// TIA Portal V15.1 export
// export: Created 2024-05-17T05:38:35.0496997Z, ExportSetting WithDefaults, DisplayName Totally Integrated Automation Portal, DisplayVersion V15.1 Update 5, DisplayName TIA Portal Openness, DisplayVersion V15.1 Update 5, DisplayName SINAMICS Startdrive Advanced, DisplayVersion V15.1, DisplayName G130, G150, S120, S150, SINAMICS MV, S210, DisplayVersion V15.1, DisplayName G110M, G120, G120C, G120D, G120P, DisplayVersion V15.1, DisplayName STEP 7 Professional, DisplayVersion V15.1 Update 5, DisplayName STEP 7 Safety, DisplayVersion V15.1, DisplayName WinCC Professional, DisplayVersion V15.1 Update 5, DisplayName SIMATIC Visualization Architect, DisplayVersion V15.1
FUNCTION_BLOCK "LProcPid"   // FB1713, FBD
TITLE = LProcPid
{ S7_Optimized_Access := 'FALSE' }
AUTHOR : VCC
FAMILY : ProcEq
NAME : Pid
VERSION : 0.1
// ================================================================================
// The Process Value is controlled by the Pid controller.
// ================================================================================
// stored: AutoNumber false, IsIECCheckEnabled false, SetENOAutomatically False, UDAEnableTagReadback false
   VAR_INPUT
      I_CYCLE { ExternalAccessible := 'False'; ExternalVisible := 'False'; ExternalWritable := 'False'} : Time;   // Sample time
      H_TI : Time;   // Pid Reset time
      H_TD : Time;   // Pid Derivative time
      I_Manual_Value { ExternalAccessible := 'False'; ExternalVisible := 'False'; ExternalWritable := 'False'} : Real;   // Pid Setpoint Manual
      I_SP_Auto : Real;   // Pid Setpoint for controller
      I_PV_PID : Real;   // Pid Process value
      H_GAIN : Real;   // Pid Proportional Gain
      H_DEADB_W : Real;   // Pid Deadband width
      H_LMN_HLM : Real := 100.0;   // Pid Manipulated value high limit
      H_LMN_LLM : Real;   // Pid Manipulated value low limit
      I_COM_RST { ExternalAccessible := 'False'; ExternalVisible := 'False'; ExternalWritable := 'False'} : Bool;   // Initialising reset of controller
      I_MAN_ON { ExternalAccessible := 'False'; ExternalVisible := 'False'; ExternalWritable := 'False'} : Bool;   // Pid Manual value on
      H_Direct : Bool := TRUE;   // Pid in Direct mode (output increase if SP>PV)
      H_P_SEL : Bool;   // Pid P selected
      H_I_SEL : Bool;   // Pid I selected
      H_D_SEL : Bool;   // Pid D selected
   END_VAR
   VAR_OUTPUT
      O_SP_PID : Real;   // Setpoint used in Pid controller
      O_LMN_PID : Real;   // Output value Pid Controller
   END_VAR
   VAR DB_SPECIFIC
      Gain { ExternalAccessible := 'False'; ExternalVisible := 'False'; ExternalWritable := 'False'} : Real;   // Pid Gain in function of Pid direct or not
      DirectCoef { ExternalAccessible := 'False'; ExternalVisible := 'False'; ExternalWritable := 'False'} : Real;   // Value +1 or -1 if Pid direct or not
      M_LMN { ExternalAccessible := 'False'; ExternalVisible := 'False'; ExternalWritable := 'False'} : Real;   // Pid Manipulated value from controller
   END_VAR
   VAR
      PidControl { ExternalAccessible := 'False'; ExternalVisible := 'False'; ExternalWritable := 'False'; S7_SetPoint := 'True'} : CONT_C;   // Pid Controller
   END_VAR
BEGIN

REGION Network 1: **** 7 - Submodules - Non-machine **** Pid control Direct: Gain>0 and Output increase when SP>PV
   // Pid control Direct: Gain>0 and Output increase when SP>PV
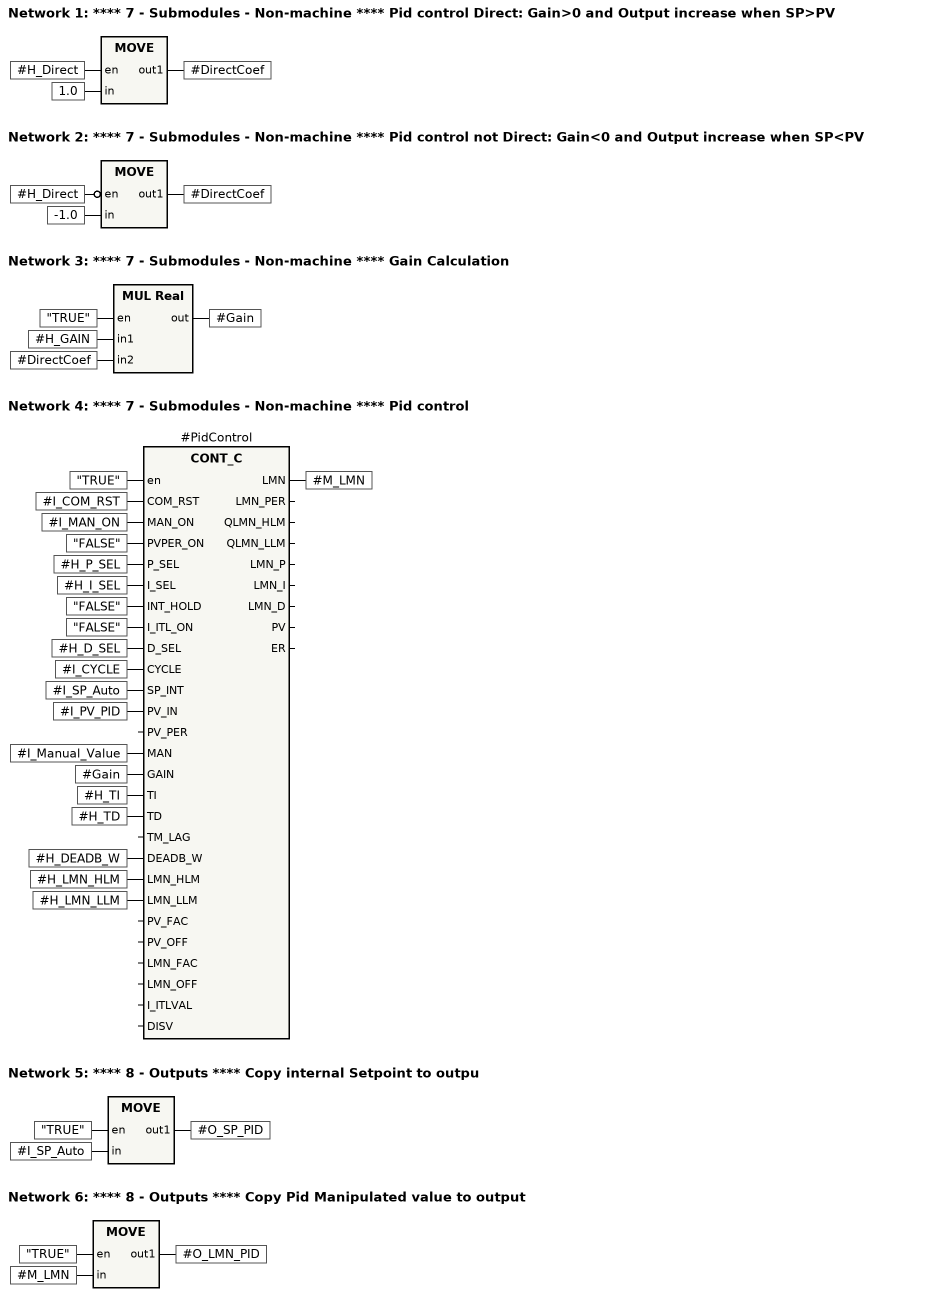
   IF #H_Direct THEN #DirectCoef := 1.0; END_IF;
END_REGION

REGION Network 2: **** 7 - Submodules - Non-machine **** Pid control not Direct: Gain<0 and Output increase when SP<PV
   // Pid control not Direct: Gain<0 and Output increase when SP<PV
   IF NOT #H_Direct THEN #DirectCoef := -1.0; END_IF;
END_REGION

REGION Network 3: **** 7 - Submodules - Non-machine **** Gain Calculation
   // Gain Calculation
   IF "TRUE" THEN #Gain := #H_GAIN * #DirectCoef; END_IF;
END_REGION

REGION Network 4: **** 7 - Submodules - Non-machine **** Pid control
   // Pid control
   IF "TRUE" THEN
       #PidControl(COM_RST := #I_COM_RST,   // CONT_C
                   MAN_ON := #I_MAN_ON,
                   PVPER_ON := "FALSE",
                   P_SEL := #H_P_SEL,
                   I_SEL := #H_I_SEL,
                   INT_HOLD := "FALSE",
                   I_ITL_ON := "FALSE",
                   D_SEL := #H_D_SEL,
                   CYCLE := #I_CYCLE,
                   SP_INT := #I_SP_Auto,
                   PV_IN := #I_PV_PID,
                   MAN := #I_Manual_Value,
                   GAIN := #Gain,
                   TI := #H_TI,
                   TD := #H_TD,
                   DEADB_W := #H_DEADB_W,
                   LMN_HLM := #H_LMN_HLM,
                   LMN_LLM := #H_LMN_LLM,
                   LMN => #M_LMN);
   END_IF;
END_REGION

REGION Network 5: **** 8 - Outputs **** Copy internal Setpoint to outpu
   // Copy internal Setpoint to output
   IF "TRUE" THEN #O_SP_PID := #I_SP_Auto; END_IF;
END_REGION

REGION Network 6: **** 8 - Outputs **** Copy Pid Manipulated value to output
   // Copy Pid Manipulated value to output
   IF "TRUE" THEN #O_LMN_PID := #M_LMN; END_IF;
END_REGION
END_FUNCTION_BLOCK
